PROGRAM C02_PCM
VAR
	fbSeqCtrl						: FB_SYSTEM_SeqControl;
	nSeqStep						: INT;

	b00_Init						: BOOL;
	b01_Idle						: BOOL;
	b03_GetNewFile				: BOOL;
	b04_ReadFile					: BOOL;
	b05_Validate					: BOOL;
	b07_Archive					: BOOL;
	b19_InitLoadDone				: BOOL;
	b20_ErrorPCMLoad				: BOOL;

	bActivatePCM					: BOOL;
	bInitLoad						: BOOL;
	bCurrentFileOverWrittenDone		: BOOL;
	bFileNotFound					: BOOL;
	bReadError					: BOOL;


	tonStartupDelay				: TON;
	fbTimer						: TON;
	rtrigReceivePCMManually		: R_TRIG;

	fbGetNewFileInfo				 : FB_FILE_GetFileInfo;
	fbReadFile					: FB_PCM_ReadFile;
	fbValidate						: FB_PCM_Validate;
	fbArchiveFile					: FB_FILE_MoveWithDate;
	fbSetLastDataToPCM				: FB_PCM_SetData;

	bValid						: BOOL;
	strFieldName					: STRING(39);
	strFieldData					: STRING(91);
	strArchiveFolder				: STRING(8);

	sPCMData_Modified				: ST_PCM_Data;
END_VAR
VAR // added by the converter: edge detectors and wires of the graphical bodies
    _w1 : BOOL;
END_VAR

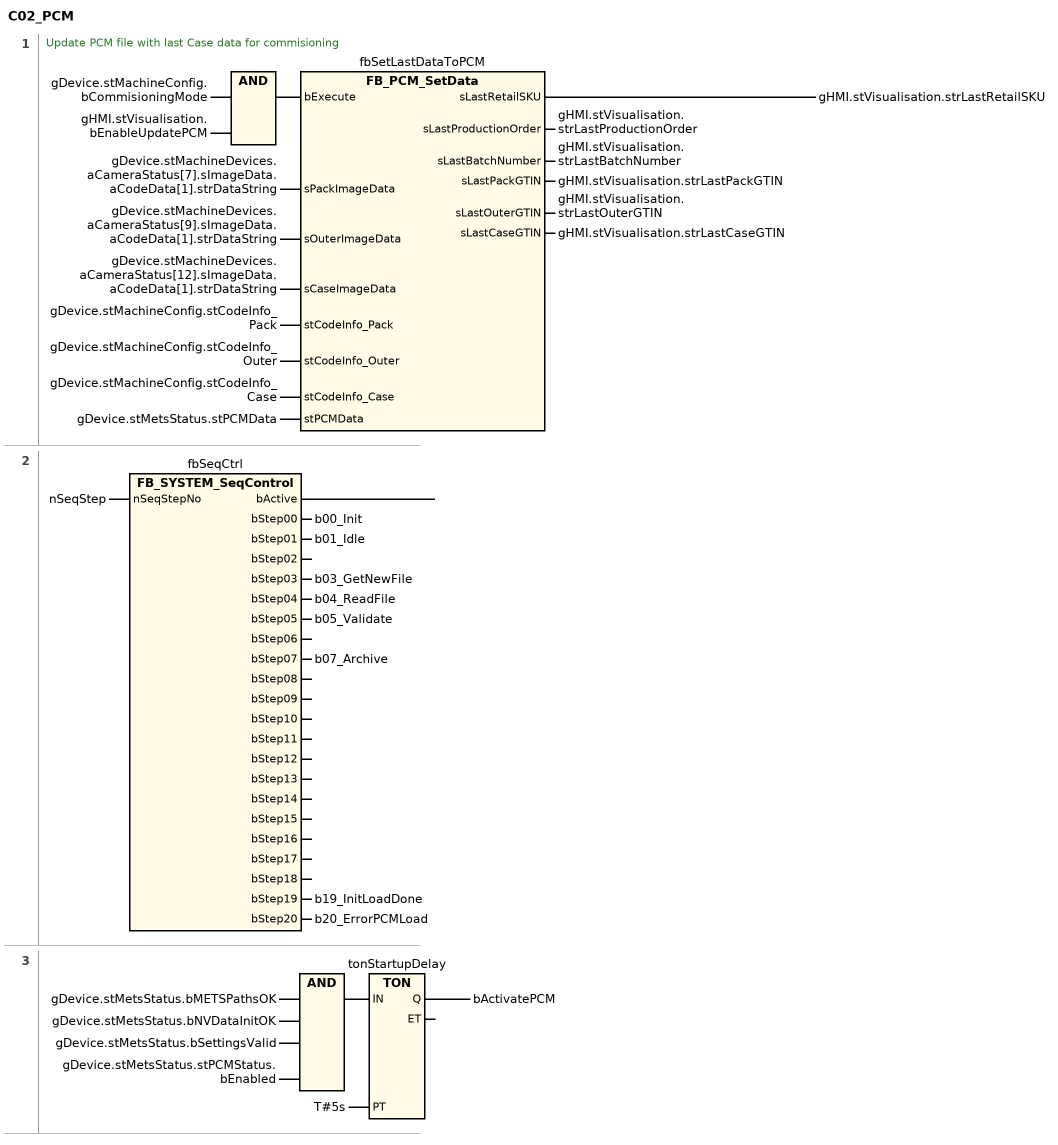
// NETWORK 1
// Update PCM file with last Case data for commisioning
fbSetLastDataToPCM(
    bExecute := gDevice.stMachineConfig.bCommisioningMode AND gHMI.stVisualisation.bEnableUpdatePCM,
    sPackImageData := gDevice.stMachineDevices.aCameraStatus[7].sImageData.aCodeData[1].strDataString,
    sOuterImageData := gDevice.stMachineDevices.aCameraStatus[9].sImageData.aCodeData[1].strDataString,
    sCaseImageData := gDevice.stMachineDevices.aCameraStatus[12].sImageData.aCodeData[1].strDataString,
    stCodeInfo_Pack := gDevice.stMachineConfig.stCodeInfo_Pack,
    stCodeInfo_Outer := gDevice.stMachineConfig.stCodeInfo_Outer,
    stCodeInfo_Case := gDevice.stMachineConfig.stCodeInfo_Case,
    stPCMData := gDevice.stMetsStatus.stPCMData,
    sLastProductionOrder => gHMI.stVisualisation.strLastProductionOrder,
    sLastBatchNumber => gHMI.stVisualisation.strLastBatchNumber,
    sLastPackGTIN => gHMI.stVisualisation.strLastPackGTIN,
    sLastOuterGTIN => gHMI.stVisualisation.strLastOuterGTIN,
    sLastCaseGTIN => gHMI.stVisualisation.strLastCaseGTIN); // FB_PCM_SetData
gHMI.stVisualisation.strLastRetailSKU := fbSetLastDataToPCM.sLastRetailSKU;

// NETWORK 2
fbSeqCtrl(
    nSeqStepNo := nSeqStep,
    bStep00 => b00_Init,
    bStep01 => b01_Idle,
    bStep03 => b03_GetNewFile,
    bStep04 => b04_ReadFile,
    bStep05 => b05_Validate,
    bStep07 => b07_Archive,
    bStep19 => b19_InitLoadDone,
    bStep20 => b20_ErrorPCMLoad); // FB_SYSTEM_SeqControl

// NETWORK 3
tonStartupDelay(IN := gDevice.stMetsStatus.bMETSPathsOK AND gDevice.stMetsStatus.bNVDataInitOK AND gDevice.stMetsStatus.bSettingsValid AND gDevice.stMetsStatus.stPCMStatus.bEnabled, PT := T#5s); // TON
bActivatePCM := tonStartupDelay.Q;

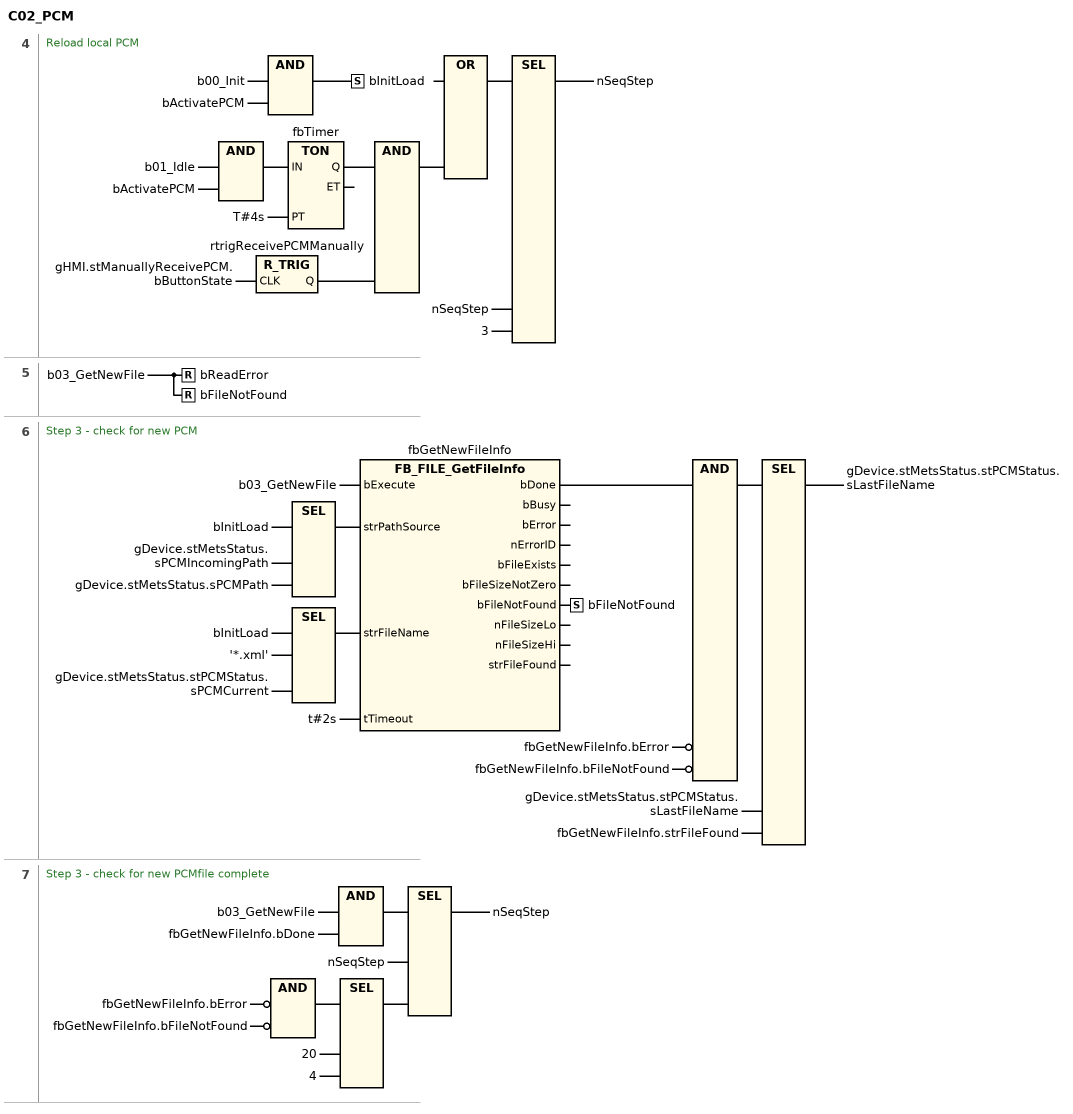
// NETWORK 4
// Reload local PCM
_w1 := b00_Init AND bActivatePCM;
bInitLoad S= _w1;
fbTimer(IN := b01_Idle AND bActivatePCM, PT := T#4s); // TON
rtrigReceivePCMManually(CLK := gHMI.stManuallyReceivePCM.bButtonState); // R_TRIG
nSeqStep := SEL(_w1 OR fbTimer.Q AND rtrigReceivePCMManually.Q, nSeqStep, 3);

// NETWORK 5
bReadError R= b03_GetNewFile;
bFileNotFound R= b03_GetNewFile;

// NETWORK 6
// Step 3 - check for new PCM
fbGetNewFileInfo(
    bExecute := b03_GetNewFile,
    strPathSource := SEL(bInitLoad, gDevice.stMetsStatus.sPCMIncomingPath, gDevice.stMetsStatus.sPCMPath),
    strFileName := SEL(bInitLoad, '*.xml', gDevice.stMetsStatus.stPCMStatus.sPCMCurrent),
    tTimeout := t#2s); // FB_FILE_GetFileInfo
bFileNotFound S= fbGetNewFileInfo.bFileNotFound;
gDevice.stMetsStatus.stPCMStatus.sLastFileName := SEL(fbGetNewFileInfo.bDone AND NOT fbGetNewFileInfo.bError AND NOT fbGetNewFileInfo.bFileNotFound, gDevice.stMetsStatus.stPCMStatus.sLastFileName, fbGetNewFileInfo.strFileFound);

// NETWORK 7
// 					Step 3 - check for new PCMfile complete
//
//
nSeqStep := SEL(b03_GetNewFile AND fbGetNewFileInfo.bDone, nSeqStep, SEL(NOT fbGetNewFileInfo.bError AND NOT fbGetNewFileInfo.bFileNotFound, 20, 4));

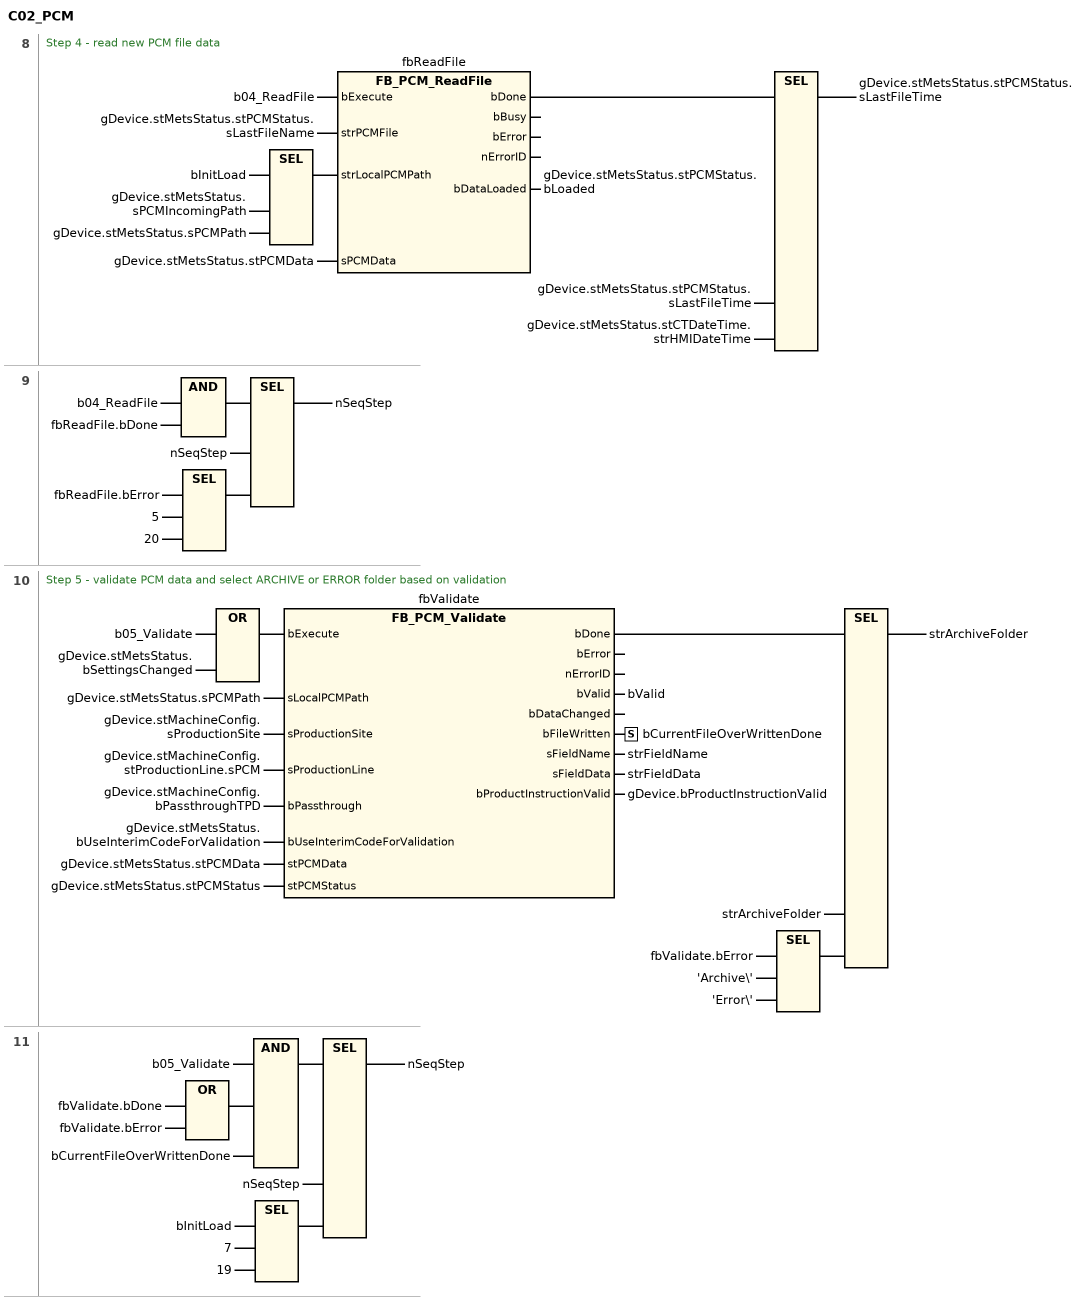
// NETWORK 8
// Step 4 - read new PCM file data
fbReadFile(
    bExecute := b04_ReadFile,
    strPCMFile := gDevice.stMetsStatus.stPCMStatus.sLastFileName,
    strLocalPCMPath := SEL(bInitLoad, gDevice.stMetsStatus.sPCMIncomingPath, gDevice.stMetsStatus.sPCMPath),
    sPCMData := gDevice.stMetsStatus.stPCMData,
    bDataLoaded => gDevice.stMetsStatus.stPCMStatus.bLoaded); // FB_PCM_ReadFile
gDevice.stMetsStatus.stPCMStatus.sLastFileTime := SEL(fbReadFile.bDone, gDevice.stMetsStatus.stPCMStatus.sLastFileTime, gDevice.stMetsStatus.stCTDateTime.strHMIDateTime);

// NETWORK 9
nSeqStep := SEL(b04_ReadFile AND fbReadFile.bDone, nSeqStep, SEL(fbReadFile.bError, 5, 20));

// NETWORK 10
// 					Step 5 - validate PCM data and select ARCHIVE or ERROR folder based on validation
//
//
fbValidate(
    bExecute := b05_Validate OR gDevice.stMetsStatus.bSettingsChanged,
    sLocalPCMPath := gDevice.stMetsStatus.sPCMPath,
    sProductionSite := gDevice.stMachineConfig.sProductionSite,
    sProductionLine := gDevice.stMachineConfig.stProductionLine.sPCM,
    bPassthrough := gDevice.stMachineConfig.bPassthroughTPD,
    bUseInterimCodeForValidation := gDevice.stMetsStatus.bUseInterimCodeForValidation,
    stPCMData := gDevice.stMetsStatus.stPCMData,
    stPCMStatus := gDevice.stMetsStatus.stPCMStatus,
    bValid => bValid,
    sFieldName => strFieldName,
    sFieldData => strFieldData,
    bProductInstructionValid => gDevice.bProductInstructionValid); // FB_PCM_Validate
bCurrentFileOverWrittenDone S= fbValidate.bFileWritten;
strArchiveFolder := SEL(fbValidate.bDone, strArchiveFolder, SEL(fbValidate.bError, 'Archive\', 'Error\'));

// NETWORK 11
nSeqStep := SEL(b05_Validate AND (fbValidate.bDone OR fbValidate.bError) AND bCurrentFileOverWrittenDone, nSeqStep, SEL(bInitLoad, 7, 19));

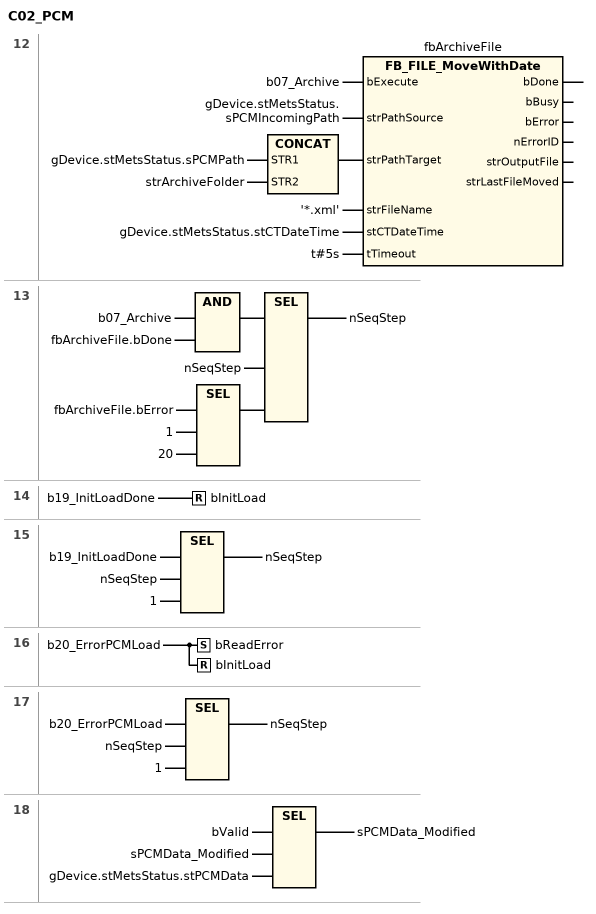
// NETWORK 12
fbArchiveFile(
    bExecute := b07_Archive,
    strPathSource := gDevice.stMetsStatus.sPCMIncomingPath,
    strPathTarget := CONCAT(STR1 := gDevice.stMetsStatus.sPCMPath, STR2 := strArchiveFolder),
    strFileName := '*.xml',
    stCTDateTime := gDevice.stMetsStatus.stCTDateTime,
    tTimeout := t#5s); // FB_FILE_MoveWithDate

// NETWORK 13
nSeqStep := SEL(b07_Archive AND fbArchiveFile.bDone, nSeqStep, SEL(fbArchiveFile.bError, 1, 20));

// NETWORK 14
bInitLoad R= b19_InitLoadDone;

// NETWORK 15
nSeqStep := SEL(b19_InitLoadDone, nSeqStep, 1);

// NETWORK 16
bReadError S= b20_ErrorPCMLoad;
bInitLoad R= b20_ErrorPCMLoad;

// NETWORK 17
nSeqStep := SEL(b20_ErrorPCMLoad, nSeqStep, 1);

// NETWORK 18
sPCMData_Modified := SEL(bValid, sPCMData_Modified, gDevice.stMetsStatus.stPCMData);

END_PROGRAM

(* stored: Version 1.1.0.1
   POU C02_PCM: Id {b5c036ef-ce0f-4502-aac5-2ffa797144fe}, SpecialFunc None *)
